// Type alias for a generic type, __SYSTEM.AnyType.
TYPE T_Generic : __SYSTEM.AnyType; END_TYPE

(* stored: Version 1.1.0.1
   DUT T_Generic: Id {6998d273-a506-0331-1179-2cc39f3b4099} *)
